// TIA Portal V17 export
// export: Created 2023-12-22T15:05:35.2939458Z, ExportSetting WithDefaults, DisplayName Totally Integrated Automation Portal, DisplayVersion V17, DisplayName TIA Portal Openness, DisplayVersion V17, DisplayName TIA Portal Version Control Interface, DisplayVersion V17, DisplayName STEP 7 Professional, DisplayVersion V17, DisplayName STEP 7 Safety, DisplayVersion V17, DisplayName WinCC Advanced, DisplayVersion V17
TYPE "In_MDA"
// stored: IsFailsafeCompliant false
   STRUCT
      CMD : Struct   // Основные команды / Блок команд
         Hand : Bool;   // 0 - авто, 1 - ручной / 0 - Авто, 1 - Ручной
         Start_A : Bool;   // Автозапуск / Запуск в авторежиме
         Start_M : Bool;   // Ручной - вперёд / Запуск в ручном режиме
         Force : Bool;   // Принудительный
         Lock : Bool;   // Блокировать / Блокировка
         Local : Bool;   // Локальный
         Service : Bool;   // Сервис
         Safety : Bool;   // Безопасность
         Alarm : Bool;   // Есть авария / Авария
         Reset : Bool;   // Сброс аварий
         Sim : Bool;   // Режим симуляции
         Vector : Bool;   // Выбор направления
         Ready : Bool;   // Разрешение дистанционного управления
         Resourse : Bool;
      END_STRUCT;
      T_ON : Int;   // Время запуска/открытия
      T_OFF : Int;   // Время останова/закрытия
      SP_M : Real;   // Задание скорости
      Converter : Struct   // Масштабирование сигнала
         Min_Out { S7_SetPoint := 'True'} : Real;   // Минимальный выходной сигнал
         Max_Out { S7_SetPoint := 'True'} : Real := 100.0;   // Максимальный выходной сигнал
      END_STRUCT;
   END_STRUCT;
END_TYPE
